FUNCTION_BLOCK E_TABLE
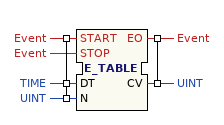
  EVENT_INPUT
    START WITH DT, N;
    STOP;
  END_EVENT
  EVENT_OUTPUT
    EO WITH CV;
  END_EVENT
  VAR_INPUT
    DT : TIME;
    N : UINT;
  END_VAR
  VAR_OUTPUT
    CV : UINT;
  END_VAR
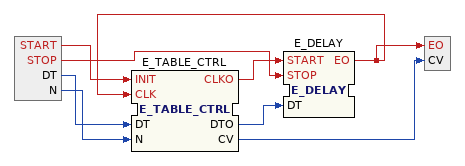
  FBS
    E_TABLE_CTRL : E_TABLE_CTRL;
    E_DELAY : E_DELAY;
  END_FBS
  EVENT_CONNECTIONS
    E_TABLE_CTRL.CLKO TO E_DELAY.START;
    E_DELAY.EO TO EO;
    START TO E_TABLE_CTRL.INIT;
    E_DELAY.EO TO E_TABLE_CTRL.CLK;
    STOP TO E_DELAY.STOP;
  END_CONNECTIONS
  DATA_CONNECTIONS
    E_TABLE_CTRL.DTO TO E_DELAY.DT;
    E_TABLE_CTRL.CV TO CV;
    DT TO E_TABLE_CTRL.DT;
    N TO E_TABLE_CTRL.N;
  END_CONNECTIONS
END_FUNCTION_BLOCK
